# B&R Automation Studio project Test01_Version_Control
Automation Studio 4.11.3.51 SP

## Configuration Config1

CPU X20CP1586, AutomationRuntime B4.92, Build 4.1.2, Vc V4.72.5

### Hardware
```
X20CP1586 : X20CP1586 v1.10.0.0
  Connector IF2:
    ActivateDevice = 1
  ConfigurationID = Test01_Version_Control_Config1
  Simulation = 1
  FileDevice1
  FileDeviceName1 = USER
  FileDevicePath1 = USER_PATH
```

## Logical view

### Global.var
```iecst
VAR
	BtnStart : BOOL;
	BtnForward : BOOL
	BtnReverse : BOOL;
	BtnStop : BOOL;
	BtnEmStop : BOOL;
	MotorConveyor : BOOL;
	MotorConveyorReverse : BOOL;
	MotorRotor : BOOL;
	MotorStator : BOOL;
	doMotorOffState : BOOL;
END_VAR
```

### Program Logical/Program

#### Main.st
```iecst
PROGRAM _INIT
	(* Insert code here *)

	//BtnStart : BOOL;
//	BtnStop : BOOL;
	//MotorConveyor : BOOL;

END_PROGRAM

PROGRAM _CYCLIC
	(* Insert code here *)

	IF BtnStart THEN
		MotorConveyor := TRUE;
	ELSIF BtnStop THEN
		MotorConveyor := FALSE;
	END_IF

END_PROGRAM

PROGRAM _EXIT
	(* Insert code here *)
//	IF BtnStop THEN
	//	MotorConveyor := FALSE;
//	END_IF

END_PROGRAM
```
